// TIA Portal V19 export
TYPE "LEXCHANGETRAY_typeSinaInput"
// stored: Access Published
   STRUCT
      enable : Bool;
      parentReferenceDesignator : WString[128];
      interlock : Bool;
      hwID : HW_IO;
      enableManualCmds : Bool;
      reset : Bool;
   END_STRUCT;
END_TYPE
